// TIA Portal project "AWL LIBRO 10" (V11)

(* hardware
DEVICE "S7300/ET200 station_1"  SIMATIC 300-Station
   slot 0: "Perfil soporte_0"  Rail  6ES7 390-1***0-0AA0
   slot 2: "PLC_1"  CPU 313C-2 DP  6ES7 313-6CF03-0AB0  V2.6
      slot 0: "Interfaz MPI_1"  MPI
      slot 1: "Interfaz DP_1"  DP
      slot 2: "DI16/DO16_1"  DI16/DO16
      slot 4: "Contaje_1"  Counter
*)

// ===== PLC "PLC_1"  CPU 313C-2 DP =====

VAR_GLOBAL   // PLC tag table "Tabla de variables estándar"
   "EMERGENCIA" AT %E0.0 : Bool;
   "MARCHA" AT %E0.1 : Bool;
   "S1" AT %E0.2 : Bool;
   "S2" AT %E0.3 : Bool;
   "S3" AT %E0.4 : Bool;
   "S4" AT %E0.5 : Bool;
   "S5" AT %E0.6 : Bool;
   "LED REPOSO" AT %A0.0 : Bool;
   "LED MARCHA / RUN" AT %A0.1 : Bool;
   "Y1 ELECTROVALVULA" AT %A0.2 : Bool;
   "Y2 ELECTROVALVULA" AT %A0.3 : Bool;
   "RESISTENCIAS CALDERA 1" AT %A0.4 : Bool;
   "Y3 ELECTROVALVULA" AT %A0.5 : Bool;
   "Y4 ELECTROVALVULA" AT %A0.6 : Bool;
   "RESISTENCIAS CALDERA 2" AT %A0.7 : Bool;
   "BATIDORA LINEA" AT %A1.0 : Bool;
   "BATIDORA ESTRELLA" AT %A1.1 : Bool;
   "BATIDORA  TRINGULO" AT %A1.2 : Bool;
   "TERMOSTATO 1" AT %E0.7 : Bool;
   "TERMOSTATO 2" AT %E1.0 : Bool;
   "SALIDAS E-VALVULAS CALDERA 1" AT %AB0 : Byte;
   "SALIDAS E-VALVULAS CALDERA 2" AT %AB1 : Byte;
   "CONTROL E-VALVULAS CALDERA 1" AT %MB0 : Byte;
   "CONTROL E-VALVULAS CALDERA 2" AT %MB1 : Byte;
   "Tag_1" AT %M0.0 : Bool;
   "Tag_2" AT %M0.1 : Bool;
   "Tag_3" AT %M0.2 : Bool;
   "Tag_4" AT %M0.3 : Bool;
   "Tag_5" AT %M0.4 : Bool;
   "Tag_6" AT %M0.5 : Bool;
   "Tag_7" AT %M0.6 : Bool;
   "Tag_8" AT %M0.7 : Bool;
   "Tag_9" AT %M1.0 : Bool;
   "Tag_10" AT %M1.1 : Bool;
   "Tag_11" AT %M1.2 : Bool;
   "SALIDAS BATIDORA" AT %AB2 : Byte;
   "CONTROL BATIDORA" AT %MB2 : Byte;
   "Tag_12" AT %M1.3 : Bool;
   "Tag_13" AT %M2.0 : Bool;
   "Tag_14" AT %M2.1 : Bool;
   "Tag_15" AT %M2.2 : Bool;
   "Y5 ELECTROVALVULA" AT %A1.3 : Bool;
   "Tag_16" AT %M2.3 : Bool;
   "Tag_17" AT %A1.4 : Bool;
   "Tag_18" AT %M1.4 : Bool;
   "Tag_19" AT %M1.7 : Bool;
   "T0" AT %T0 : Timer;
   "T1" AT %T1 : Timer;
END_VAR

DATA_BLOCK "F Y B"   // DB1
{ S7_Optimized_Access := 'FALSE' }
VERSION : 0.1
   VAR
      F0 : Bool;
      F1 : Bool;
      F2 : Bool;
      F3 : Bool;
      F4 : Bool;
      F5 : Bool;
      F6 : Bool;
      F7 : Bool;
      B0 : Bool;
      B1 : Bool;
      B3 : Bool;
   END_VAR
BEGIN
END_DATA_BLOCK

ORGANIZATION_BLOCK "Main"   // OB1, STL
TITLE = EJERCICIO 10 / "Main Program Sweep (Cycle)"
{ S7_Optimized_Access := 'FALSE' }
VERSION : 0.1
   VAR_TEMP
      OB1_EV_CLASS : Byte;   // Bits 0-3 = 1 (Coming event), Bits 4-7 = 1 (Event class 1)
      OB1_SCAN_1 : Byte;   // 1 (Cold restart scan 1 of OB 1), 3 (Scan 2-n of OB 1)
      OB1_PRIORITY : Byte;   // Priority of OB Execution
      OB1_OB_NUMBR : Byte;   // 1 (Organization block 1, OB1)
      OB1_RESERVED_1 : Byte;   // Reserved for system
      OB1_RESERVED_2 : Byte;   // Reserved for system
      OB1_PREV_CYCLE : Int;   // Cycle time of previous OB1 scan (milliseconds)
      OB1_MIN_CYCLE : Int;   // Minimum cycle time of OB1 (milliseconds)
      OB1_MAX_CYCLE : Int;   // Maximum cycle time of OB1 (milliseconds)
      OB1_DATE_TIME : Date_And_Time;   // Date and time OB1 started
   END_VAR
BEGIN
END_ORGANIZATION_BLOCK